FUNCTION_BLOCK PUBLIC FB_MusicPlayCommand IMPLEMENTS I_Command
VAR
	refCDPlayer : REFERENCE TO FB_CDPlayer;
END_VAR

METHOD Execute
IF (__ISVALIDREF(THIS^.refCDPlayer)) THEN
	THIS^.refCDPlayer.SetVolume(40);
	THIS^.refCDPlayer.SetTrack(1);
	THIS^.refCDPlayer.Start();
END_IF
END_METHOD

METHOD FB_init : BOOL
VAR_INPUT
	bInitRetains : BOOL; // if TRUE, the retain variables are initialized (warm start / cold start)
	bInCopyCode : BOOL;  // if TRUE, the instance afterwards gets moved into the copy code (online change)
	refCDPlayer : REFERENCE TO FB_CDPlayer;
END_VAR
IF (__ISVALIDREF(refCDPlayer)) THEN
	THIS^.refCDPlayer REF= refCDPlayer;
ELSE
	THIS^.refCDPlayer REF= 0;
END_IF
END_METHOD

METHOD Undo
IF (__ISVALIDREF(THIS^.refCDPlayer)) THEN
	THIS^.refCDPlayer.Stop();
END_IF
END_METHOD

END_FUNCTION_BLOCK

(* stored: Version 1.1.0.1, ProductVersion 3.1.4020.3
   POU FB_MusicPlayCommand: Id {9af7a132-dfd1-40f6-9e03-6c734bb23364}, SpecialFunc None
   Method Execute: Id {1e3196d6-937f-40cc-beb7-c27b776095f5}
   Method FB_init: Id {4d51c6d5-7d44-4836-8364-0806c83c0c3c}
   Method Undo: Id {0b52a410-f7bb-4718-b299-09bc3da2601e} *)
